//==================================================================================================
//							Beckhoff Automation Poland
//									19.10.2018
//	Program wykrywajacy bledy dzielnia przez 0 i przekraczania zakresow zmiennych, tablic...
// 
//	v1.4	|| TC v 3.1.4022.25		|| - Ustawiono setowanie bledow, dodano wejscie bReset 
//	v1.3	|| TC v 3.1.4022.16		|| - Przeniesiono logowanie do EventLoggera wraz z zabepieczeniem przed zbyt szybkim logowaniem zdarzeń do programu P_SystemDiag_EventLog. 
//	v1.2	|| TC v 3.1.4020.28		|| - Dodano logowanie do EventLoggera wraz z zabepieczeniem przed zbyt szybki logowaniem zdarzeń
//	v1.1 	|| TC v 3.1.4020.14 	|| - Dodane wyjscia bOk, bWarning, bError
//	v1.0 	|| TC v 3.1.4020.0 		|| - Pierwsza wersja
//==================================================================================================
PROGRAM P_Checks
VAR_INPUT
	bReset							: BOOL;
END_VAR
VAR_OUTPUT
	bOK								: BOOL;	// Brak bledow i ostrzezen
	bWarning						: BOOL;	// Ostrzezenie - nie wystepuja w tym podprogramie - wystepuja dla zachowania spojnosci
	bError							: BOOL;	// Zbiorcza flaga bledow
	udiErrorID						: UDINT;       
	sErrorDescription				: WSTRING;
END_VAR
VAR
	bCheckBounds					: BOOL;	// Flaga przekroczen zakresu indexow, np. tablic
	bCheckDivDInt					: BOOL;	// Flaga prob dzielenia Dint przez 0
	bCheckDivLInt					: BOOL; // Flaga prob dzielenia LInt przez 0
	bCheckDivLReal					: BOOL; // Flaga prob dzielenia LREAL przez 0
	bCheckDivReal					: BOOL; // Flaga prob dzielenia REAL przez 0
	bCheckRangeSigned				: BOOL;	// Flaga przekroczen liczby znakowej
	bCheckRangeUnsigned				: BOOL; // Flaga przekroczen liczby bezznakowej
	
	dCheckBoundsOld					: DINT;	// Licznik przekroczen zakresu indexow, np. tablic
	dCheckDivDIntOld				: DINT;	// Licznik prob dzielenia Dint przez 0
	dCheckDivLIntOld				: DINT; // Licznik prob dzielenia LInt przez 0
	dCheckDivLRealOld				: DINT; // Licznik prob dzielenia LREAL przez 0
	dCheckDivRealOld				: DINT; // Licznik prob dzielenia REAL przez 0
	dCheckRangeSignedOld			: DINT;	// Licznik przekroczen  liczby znakowej
	dCheckRangeUnsignedOld			: DINT; // Licznik przekroczen  liczby bezznakowej
	
	rtError							: R_TRIG;
END_VAR

IF bReset THEN
	bCheckBounds 					:= FALSE;
	bCheckDivDInt					:= FALSE;
	bCheckDivLInt					:= FALSE;
	bCheckDivLReal					:= FALSE;
	bCheckDivReal					:= FALSE;
	bCheckRangeSigned				:= FALSE;
	bCheckRangeUnsigned				:= FALSE;
ELSE
	bCheckBounds 					S= dCheckBoundsOld <> gvlChecks.dCheckBounds;
	bCheckDivDInt					S= dCheckDivDIntOld <> gvlChecks.dCheckDivDInt;
	bCheckDivLInt					S= dCheckDivLIntOld <> gvlChecks.dCheckDivLInt;
	bCheckDivLReal					S= dCheckDivLRealOld <> gvlChecks.dCheckDivLReal;
	bCheckDivReal					S= dCheckDivRealOld <> gvlChecks.dCheckDivReal;
	bCheckRangeSigned				S= dCheckRangeSignedOld <> gvlChecks.dCheckRangeSigned;
	bCheckRangeUnsigned				S= dCheckRangeUnsignedOld <> gvlChecks.dCheckRangeUnsigned;	
END_IF

dCheckBoundsOld 					:= gvlChecks.dCheckBounds;
dCheckDivDIntOld 					:= gvlChecks.dCheckDivDInt;
dCheckDivLIntOld 					:= gvlChecks.dCheckDivLInt;
dCheckDivLRealOld 					:= gvlChecks.dCheckDivLReal;
dCheckDivRealOld 					:= gvlChecks.dCheckDivReal;
dCheckRangeSignedOld 				:= gvlChecks.dCheckRangeSigned;
dCheckRangeUnsignedOld 				:= gvlChecks.dCheckRangeUnsigned;

bError 								:= bCheckBounds OR bCheckDivDInt OR bCheckDivLInt OR bCheckDivLReal OR bCheckDivReal OR bCheckRangeSigned OR bCheckRangeUnsigned;
bOK 								:= NOT bError AND NOT bWarning;


rtError								(CLK:= bError);
                                    
IF rtError.Q THEN                   
	udiErrorID						:= 99;                         
	sErrorDescription				:= "Błąd sterownika | Błąd programu sprawdzającego operacje sterownika";	
END_IF                              
                                    
IF NOT bError THEN                  
	udiErrorID						:= 0;	
	sErrorDescription				:= "";
END_IF

END_PROGRAM

(* stored: Version 1.1.0.1, ProductVersion 3.1.4026.13, FileIdentifier 6d009aaf65c2143650d3e296e3d7d9e881928667, FileSignature 9cbb7ce055127d7262ac5e67e1752651b92c5d56df09d4be4ac20337701b67f53086d31a891a650362b5f9289c310a3c15543e34f42642e8e3807d979f99a9ea6b8f6f54367612016eb67a9b48281e2bebe30a08199a40e08f34821ad0abdb91c4d3b108f9b7e9700a923c61758d34870d1879d868c92905bf3e04f478414a1861c2d2d080ab81fe4cbae8c2fc9f1cde242f41aa6b61399073a45384a88a3da92a0becf88bd1181b7736f6bf257a74a072bc52c42c79ee099a1b8a05836ab2cc251acd8c78c88beb932a6027ad0959458d48d5350abe99be1410aef7c9e8eb03cd6c4fbbdac38653d066de3b4bcf80536cde5110e719e294feb5345524ec46b3
   POU P_Checks: Id {bce355f9-21e8-41bf-a535-a57361862bad}, SpecialFunc None *)
